{attribute 'GeneratedUsingTerminal: EJ2521-0224-0016'}
{attribute addProperty BoxType "EJ2521-0224-0016"}
{attribute addProperty Id "Enable_PLSBOOL1OutputBOOL1"}
{attribute addProperty CRC "2005331871"}
{attribute addProperty Size "2"}
TYPE Control_7786EF9F :
STRUCT
	{attribute addProperty Name "Enable_PLS"}
	Enable_PLS : BOOL;
	{attribute addProperty Name "Output"}
	Output : BOOL;
END_STRUCT
END_TYPE

(* stored: Version 1.2.0.0, ProductVersion 3.1.4024.9
   DUT Control_7786EF9F: Id {24174db3-e736-45f3-ac46-b96310f04dd1} *)
